// TIA Portal V19 export
TYPE "LEXCHANGETRAY_typeHandlingXyz_signalTM_Interface"
// stored: Access Published
   STRUCT
      cmd : "LEXCHANGETRAY_typeHandlingXyz_signalTM_Cmd";
      monitor { S7_SetPoint := 'True'} : "LEXCHANGETRAY_typeHandlingXyz_signalTM_Monitor";
      sim { S7_SetPoint := 'True'} : "LEXCHANGETRAY_typeHandlingXyz_signalTM_Simulation";
   END_STRUCT;
END_TYPE
